// TIA Portal V15.1 export
// export: Created 2024-05-17T05:38:55.5007339Z, ExportSetting WithDefaults, DisplayName Totally Integrated Automation Portal, DisplayVersion V15.1 Update 5, DisplayName TIA Portal Openness, DisplayVersion V15.1 Update 5, DisplayName SINAMICS Startdrive Advanced, DisplayVersion V15.1, DisplayName G130, G150, S120, S150, SINAMICS MV, S210, DisplayVersion V15.1, DisplayName G110M, G120, G120C, G120D, G120P, DisplayVersion V15.1, DisplayName STEP 7 Professional, DisplayVersion V15.1 Update 5, DisplayName STEP 7 Safety, DisplayVersion V15.1, DisplayName WinCC Professional, DisplayVersion V15.1 Update 5, DisplayName SIMATIC Visualization Architect, DisplayVersion V15.1
FUNCTION "209220ZM01Config" : Void   // FC352, FBD
TITLE = 209220ZM01 ModeZone Configuration
{ S7_Optimized_Access := 'FALSE' }
AUTHOR : VCC
VERSION : 0.1
// stored: AutoNumber false, IsIECCheckEnabled false, SetENOAutomatically False, UDAEnableTagReadback false
BEGIN

REGION Network 1: **** 4.2 - Machine Status - Parameters **** Andon
   // Andon Config VCG
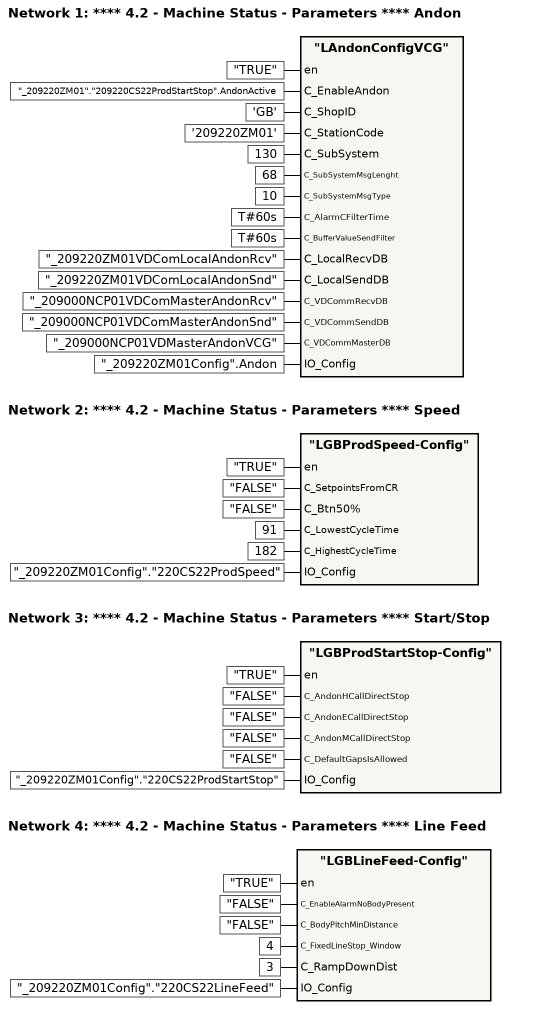
   IF "TRUE" THEN
       "LAndonConfigVCG"(C_EnableAndon := "_209220ZM01"."209220CS22ProdStartStop".AndonActive,
                         C_ShopID := 'GB',
                         C_StationCode := '209220ZM01',
                         C_SubSystem := 130,
                         C_SubSystemMsgLenght := 68,
                         C_SubSystemMsgType := 10,
                         C_AlarmCFilterTime := T#60s,
                         C_BufferValueSendFilter := T#60s,
                         C_LocalRecvDB := "_209220ZM01VDComLocalAndonRcv",
                         C_LocalSendDB := "_209220ZM01VDComLocalAndonSnd",
                         C_VDCommRecvDB := "_209000NCP01VDComMasterAndonRcv",
                         C_VDCommSendDB := "_209000NCP01VDComMasterAndonSnd",
                         C_VDCommMasterDB := "_209000NCP01VDMasterAndonVCG",
                         IO_Config := "_209220ZM01Config".Andon);
   END_IF;
END_REGION

REGION Network 2: **** 4.2 - Machine Status - Parameters **** Speed
   IF "TRUE" THEN
       "LGBProdSpeed-Config"(C_SetpointsFromCR := "FALSE",
                             "C_Btn50%" := "FALSE",
                             C_LowestCycleTime := 91,
                             C_HighestCycleTime := 182,
                             IO_Config := "_209220ZM01Config"."220CS22ProdSpeed");
   END_IF;
END_REGION

REGION Network 3: **** 4.2 - Machine Status - Parameters **** Start/Stop
   IF "TRUE" THEN
       "LGBProdStartStop-Config"(C_AndonHCallDirectStop := "FALSE",
                               C_AndonECallDirectStop := "FALSE",
                               C_AndonMCallDirectStop := "FALSE",
                               C_DefaultGapsIsAllowed := "FALSE",
                               IO_Config := "_209220ZM01Config"."220CS22ProdStartStop");
   END_IF;
END_REGION

REGION Network 4: **** 4.2 - Machine Status - Parameters **** Line Feed
   IF "TRUE" THEN
       "LGBLineFeed-Config"(C_EnableAlarmNoBodyPresent := "FALSE",
                            C_BodyPitchMinDistance := "FALSE",
                            C_FixedLineStop_Window := 4,
                            C_RampDownDist := 3,
                            IO_Config := "_209220ZM01Config"."220CS22LineFeed");
   END_IF;
END_REGION

REGION Network 5: **** 4.2 - Machine Status - Parameters **** Shift Register
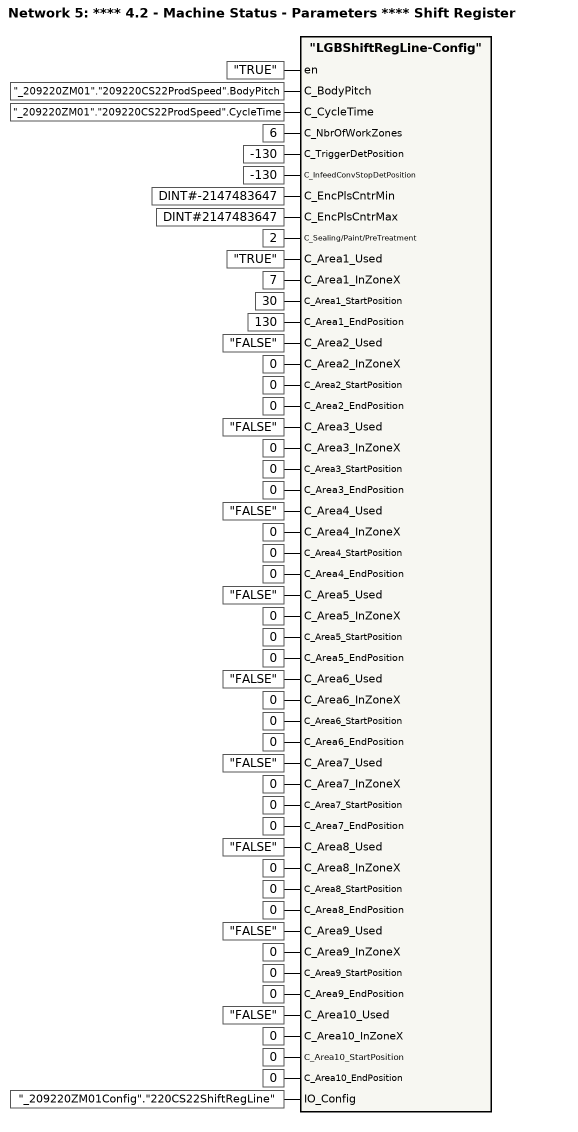
   IF "TRUE" THEN
       "LGBShiftRegLine-Config"(C_BodyPitch := "_209220ZM01"."209220CS22ProdSpeed".BodyPitch,
                               C_CycleTime := "_209220ZM01"."209220CS22ProdSpeed".CycleTime,
                               C_NbrOfWorkZones := 6,
                               C_TriggerDetPosition := -130,
                               C_InfeedConvStopDetPosition := -130,
                               C_EncPlsCntrMin := DINT#-2147483647,
                               C_EncPlsCntrMax := DINT#2147483647,
                               "C_Sealing/Paint/PreTreatment" := 2,
                               C_Area1_Used := "TRUE",
                               C_Area1_InZoneX := 7,
                               C_Area1_StartPosition := 30,
                               C_Area1_EndPosition := 130,
                               C_Area2_Used := "FALSE",
                               C_Area2_InZoneX := 0,
                               C_Area2_StartPosition := 0,
                               C_Area2_EndPosition := 0,
                               C_Area3_Used := "FALSE",
                               C_Area3_InZoneX := 0,
                               C_Area3_StartPosition := 0,
                               C_Area3_EndPosition := 0,
                               C_Area4_Used := "FALSE",
                               C_Area4_InZoneX := 0,
                               C_Area4_StartPosition := 0,
                               C_Area4_EndPosition := 0,
                               C_Area5_Used := "FALSE",
                               C_Area5_InZoneX := 0,
                               C_Area5_StartPosition := 0,
                               C_Area5_EndPosition := 0,
                               C_Area6_Used := "FALSE",
                               C_Area6_InZoneX := 0,
                               C_Area6_StartPosition := 0,
                               C_Area6_EndPosition := 0,
                               C_Area7_Used := "FALSE",
                               C_Area7_InZoneX := 0,
                               C_Area7_StartPosition := 0,
                               C_Area7_EndPosition := 0,
                               C_Area8_Used := "FALSE",
                               C_Area8_InZoneX := 0,
                               C_Area8_StartPosition := 0,
                               C_Area8_EndPosition := 0,
                               C_Area9_Used := "FALSE",
                               C_Area9_InZoneX := 0,
                               C_Area9_StartPosition := 0,
                               C_Area9_EndPosition := 0,
                               C_Area10_Used := "FALSE",
                               C_Area10_InZoneX := 0,
                               C_Area10_StartPosition := 0,
                               C_Area10_EndPosition := 0,
                               IO_Config := "_209220ZM01Config"."220CS22ShiftRegLine");
   END_IF;
END_REGION

REGION Network 6: **** 4.2 - Machine Status - Parameters **** 220CHB21
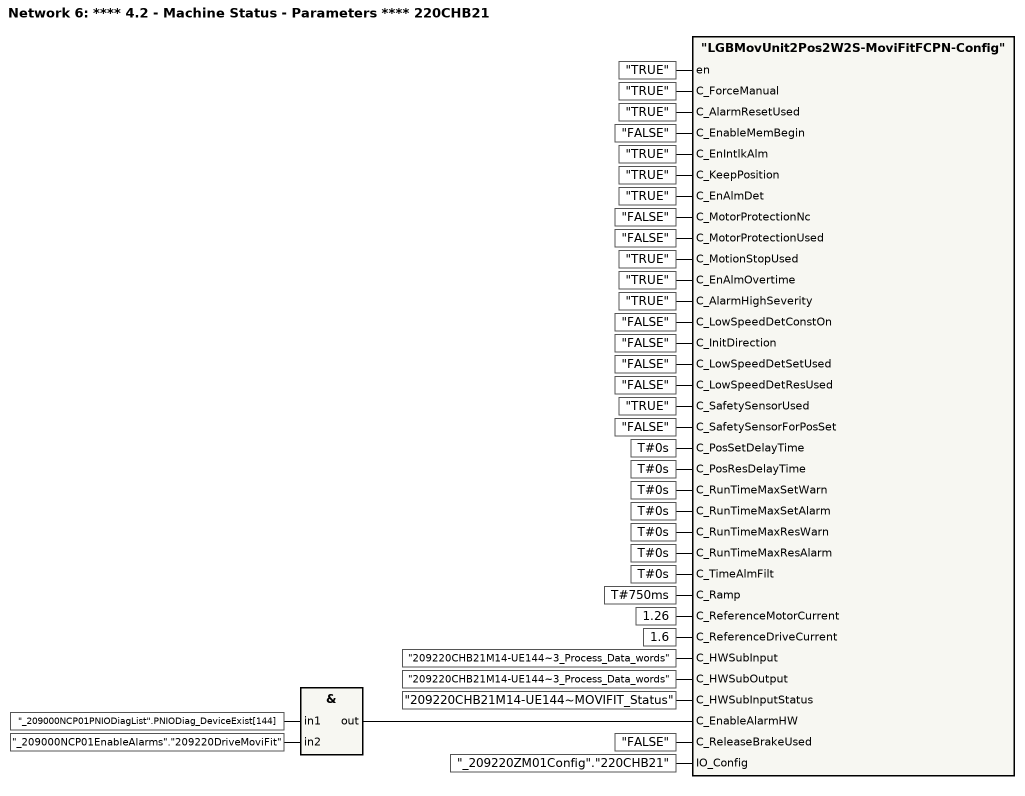
   IF "TRUE" THEN
       "LGBMovUnit2Pos2W2S-MoviFitFCPN-Config"(C_ForceManual := "TRUE",
                               C_AlarmResetUsed := "TRUE",
                               C_EnableMemBegin := "FALSE",
                               C_EnIntlkAlm := "TRUE",
                               C_KeepPosition := "TRUE",
                               C_EnAlmDet := "TRUE",
                               C_MotorProtectionNc := "FALSE",
                               C_MotorProtectionUsed := "FALSE",
                               C_MotionStopUsed := "TRUE",
                               C_EnAlmOvertime := "TRUE",
                               C_AlarmHighSeverity := "TRUE",
                               C_LowSpeedDetConstOn := "FALSE",
                               C_InitDirection := "FALSE",
                               C_LowSpeedDetSetUsed := "FALSE",
                               C_LowSpeedDetResUsed := "FALSE",
                               C_SafetySensorUsed := "TRUE",
                               C_SafetySensorForPosSet := "FALSE",
                               C_PosSetDelayTime := T#0s,
                               C_PosResDelayTime := T#0s,
                               C_RunTimeMaxSetWarn := T#0s,
                               C_RunTimeMaxSetAlarm := T#0s,
                               C_RunTimeMaxResWarn := T#0s,
                               C_RunTimeMaxResAlarm := T#0s,
                               C_TimeAlmFilt := T#0s,
                               C_Ramp := T#750ms,
                               C_ReferenceMotorCurrent := 1.26,
                               C_ReferenceDriveCurrent := 1.6,
                               C_HWSubInput := "209220CHB21M14-UE144~3_Process_Data_words",
                               C_HWSubOutput := "209220CHB21M14-UE144~3_Process_Data_words",
                               C_HWSubInputStatus := "209220CHB21M14-UE144~MOVIFIT_Status",
                               C_EnableAlarmHW := "_209000NCP01PNIODiagList".PNIODiag_DeviceExist[144] AND "_209000NCP01EnableAlarms"."209220DriveMoviFit",
                               C_ReleaseBrakeUsed := "FALSE",
                               IO_Config := "_209220ZM01Config"."220CHB21");
   END_IF;
END_REGION

REGION Network 7: **** 4.2 - Machine Status - Parameters **** 220CR21
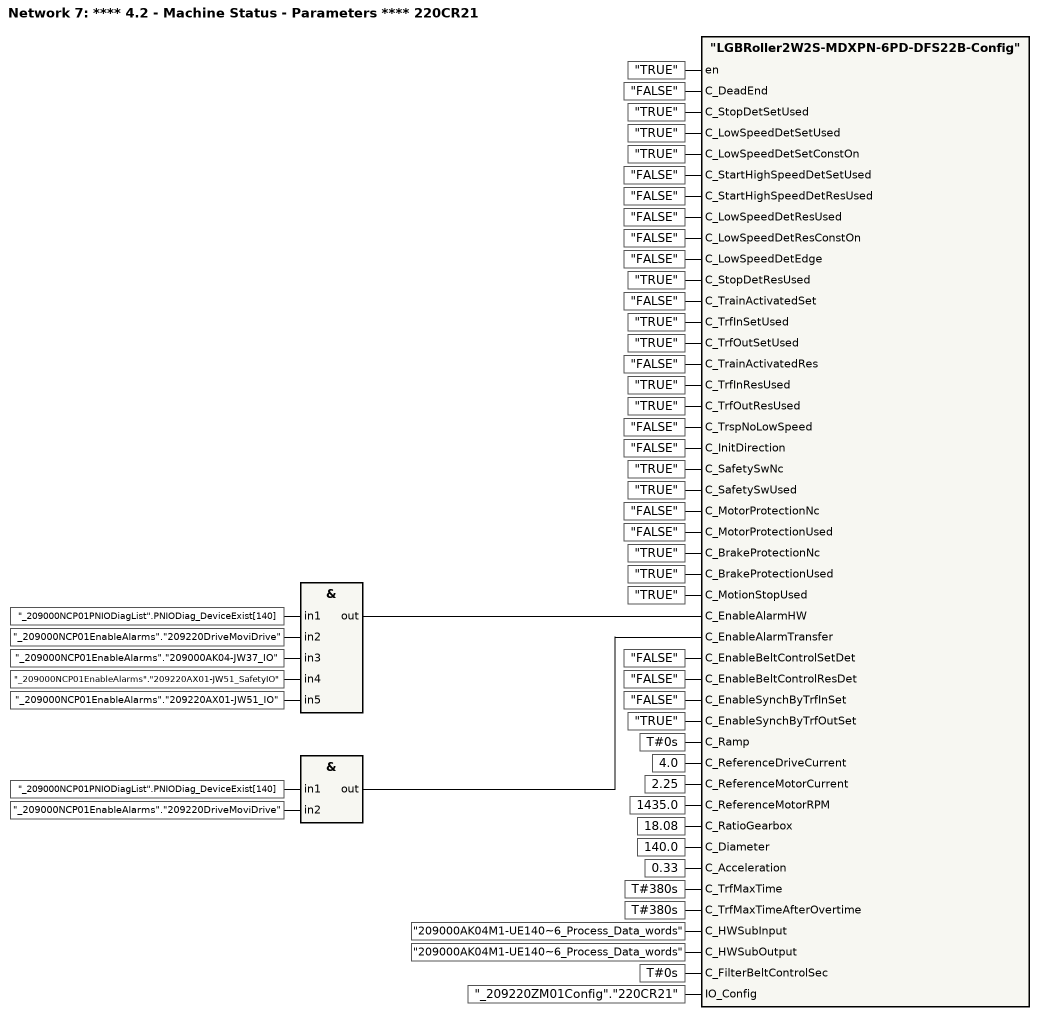
   IF "TRUE" THEN
       "LGBRoller2W2S-MDXPN-6PD-DFS22B-Config"(C_DeadEnd := "FALSE",
                               C_StopDetSetUsed := "TRUE",
                               C_LowSpeedDetSetUsed := "TRUE",
                               C_LowSpeedDetSetConstOn := "TRUE",
                               C_StartHighSpeedDetSetUsed := "FALSE",
                               C_StartHighSpeedDetResUsed := "FALSE",
                               C_LowSpeedDetResUsed := "FALSE",
                               C_LowSpeedDetResConstOn := "FALSE",
                               C_LowSpeedDetEdge := "FALSE",
                               C_StopDetResUsed := "TRUE",
                               C_TrainActivatedSet := "FALSE",
                               C_TrfInSetUsed := "TRUE",
                               C_TrfOutSetUsed := "TRUE",
                               C_TrainActivatedRes := "FALSE",
                               C_TrfInResUsed := "TRUE",
                               C_TrfOutResUsed := "TRUE",
                               C_TrspNoLowSpeed := "FALSE",
                               C_InitDirection := "FALSE",
                               C_SafetySwNc := "TRUE",
                               C_SafetySwUsed := "TRUE",
                               C_MotorProtectionNc := "FALSE",
                               C_MotorProtectionUsed := "FALSE",
                               C_BrakeProtectionNc := "TRUE",
                               C_BrakeProtectionUsed := "TRUE",
                               C_MotionStopUsed := "TRUE",
                               C_EnableAlarmHW := "_209000NCP01PNIODiagList".PNIODiag_DeviceExist[140] AND "_209000NCP01EnableAlarms"."209220DriveMoviDrive" AND "_209000NCP01EnableAlarms"."209000AK04-JW37_IO" AND "_209000NCP01EnableAlarms"."209220AX01-JW51_SafetyIO" AND "_209000NCP01EnableAlarms"."209220AX01-JW51_IO",
                               C_EnableAlarmTransfer := "_209000NCP01PNIODiagList".PNIODiag_DeviceExist[140] AND "_209000NCP01EnableAlarms"."209220DriveMoviDrive",
                               C_EnableBeltControlSetDet := "FALSE",
                               C_EnableBeltControlResDet := "FALSE",
                               C_EnableSynchByTrfInSet := "FALSE",
                               C_EnableSynchByTrfOutSet := "TRUE",
                               C_Ramp := T#0s,
                               C_ReferenceDriveCurrent := 4.0,
                               C_ReferenceMotorCurrent := 2.25,
                               C_ReferenceMotorRPM := 1435.0,
                               C_RatioGearbox := 18.08,
                               C_Diameter := 140.0,
                               C_Acceleration := 0.33,
                               C_TrfMaxTime := T#380s,
                               C_TrfMaxTimeAfterOvertime := T#380s,
                               C_HWSubInput := "209000AK04M1-UE140~6_Process_Data_words",
                               C_HWSubOutput := "209000AK04M1-UE140~6_Process_Data_words",
                               C_FilterBeltControlSec := T#0s,
                               IO_Config := "_209220ZM01Config"."220CR21");
   END_IF;
END_REGION

REGION Network 8: **** 4.2 - Machine Status - Parameters **** 220CS22
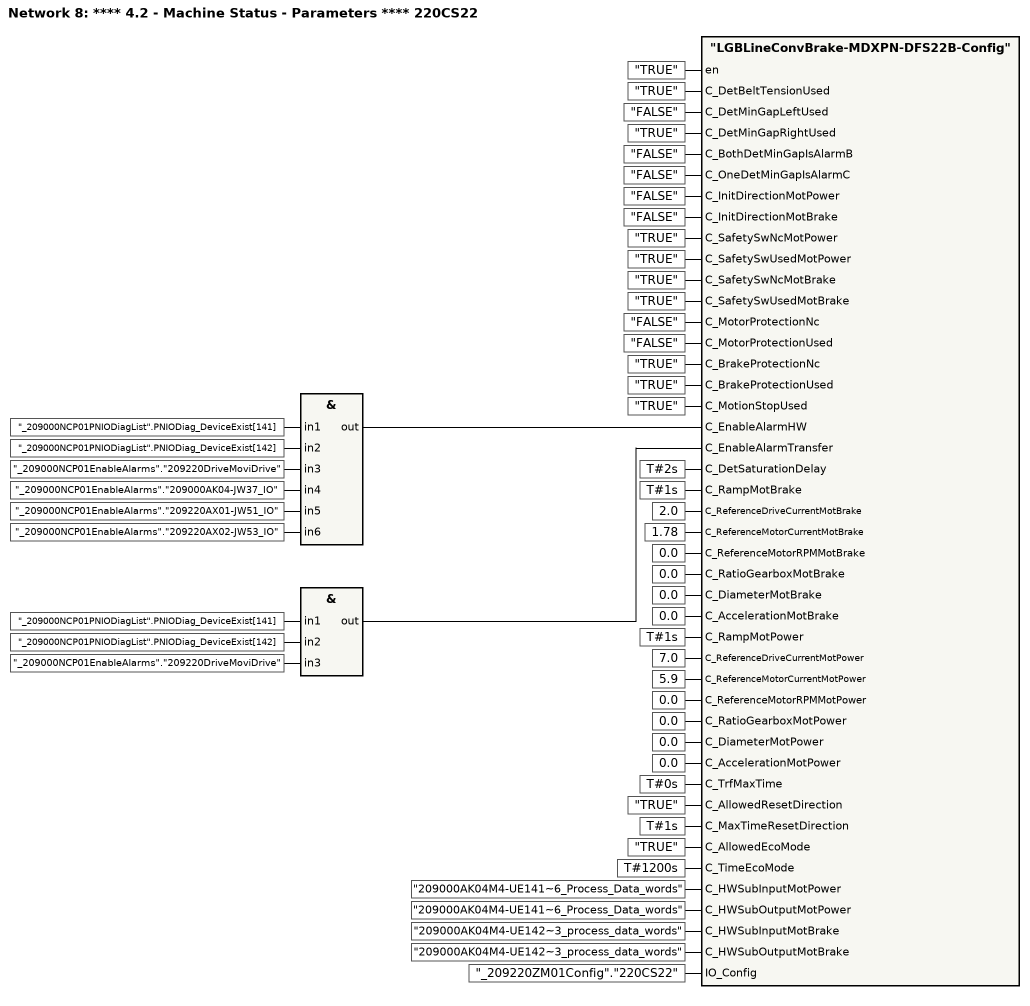
   IF "TRUE" THEN
       "LGBLineConvBrake-MDXPN-DFS22B-Config"(C_DetBeltTensionUsed := "TRUE",
                               C_DetMinGapLeftUsed := "FALSE",
                               C_DetMinGapRightUsed := "TRUE",
                               C_BothDetMinGapIsAlarmB := "FALSE",
                               C_OneDetMinGapIsAlarmC := "FALSE",
                               C_InitDirectionMotPower := "FALSE",
                               C_InitDirectionMotBrake := "FALSE",
                               C_SafetySwNcMotPower := "TRUE",
                               C_SafetySwUsedMotPower := "TRUE",
                               C_SafetySwNcMotBrake := "TRUE",
                               C_SafetySwUsedMotBrake := "TRUE",
                               C_MotorProtectionNc := "FALSE",
                               C_MotorProtectionUsed := "FALSE",
                               C_BrakeProtectionNc := "TRUE",
                               C_BrakeProtectionUsed := "TRUE",
                               C_MotionStopUsed := "TRUE",
                               C_EnableAlarmHW := "_209000NCP01PNIODiagList".PNIODiag_DeviceExist[141] AND "_209000NCP01PNIODiagList".PNIODiag_DeviceExist[142] AND "_209000NCP01EnableAlarms"."209220DriveMoviDrive" AND "_209000NCP01EnableAlarms"."209000AK04-JW37_IO" AND "_209000NCP01EnableAlarms"."209220AX01-JW51_IO" AND "_209000NCP01EnableAlarms"."209220AX02-JW53_IO",
                               C_EnableAlarmTransfer := "_209000NCP01PNIODiagList".PNIODiag_DeviceExist[141] AND "_209000NCP01PNIODiagList".PNIODiag_DeviceExist[142] AND "_209000NCP01EnableAlarms"."209220DriveMoviDrive",
                               C_DetSaturationDelay := T#2s,
                               C_RampMotBrake := T#1s,
                               C_ReferenceDriveCurrentMotBrake := 2.0,
                               C_ReferenceMotorCurrentMotBrake := 1.78,
                               C_ReferenceMotorRPMMotBrake := 0.0,
                               C_RatioGearboxMotBrake := 0.0,
                               C_DiameterMotBrake := 0.0,
                               C_AccelerationMotBrake := 0.0,
                               C_RampMotPower := T#1s,
                               C_ReferenceDriveCurrentMotPower := 7.0,
                               C_ReferenceMotorCurrentMotPower := 5.9,
                               C_ReferenceMotorRPMMotPower := 0.0,
                               C_RatioGearboxMotPower := 0.0,
                               C_DiameterMotPower := 0.0,
                               C_AccelerationMotPower := 0.0,
                               C_TrfMaxTime := T#0s,
                               C_AllowedResetDirection := "TRUE",
                               C_MaxTimeResetDirection := T#1s,
                               C_AllowedEcoMode := "TRUE",
                               C_TimeEcoMode := T#1200s,
                               C_HWSubInputMotPower := "209000AK04M4-UE141~6_Process_Data_words",
                               C_HWSubOutputMotPower := "209000AK04M4-UE141~6_Process_Data_words",
                               C_HWSubInputMotBrake := "209000AK04M4-UE142~3_process_data_words",
                               C_HWSubOutputMotBrake := "209000AK04M4-UE142~3_process_data_words",
                               IO_Config := "_209220ZM01Config"."220CS22");
   END_IF;
END_REGION

REGION Network 9: **** 4.2 - Machine Status - Parameters **** 220CR23
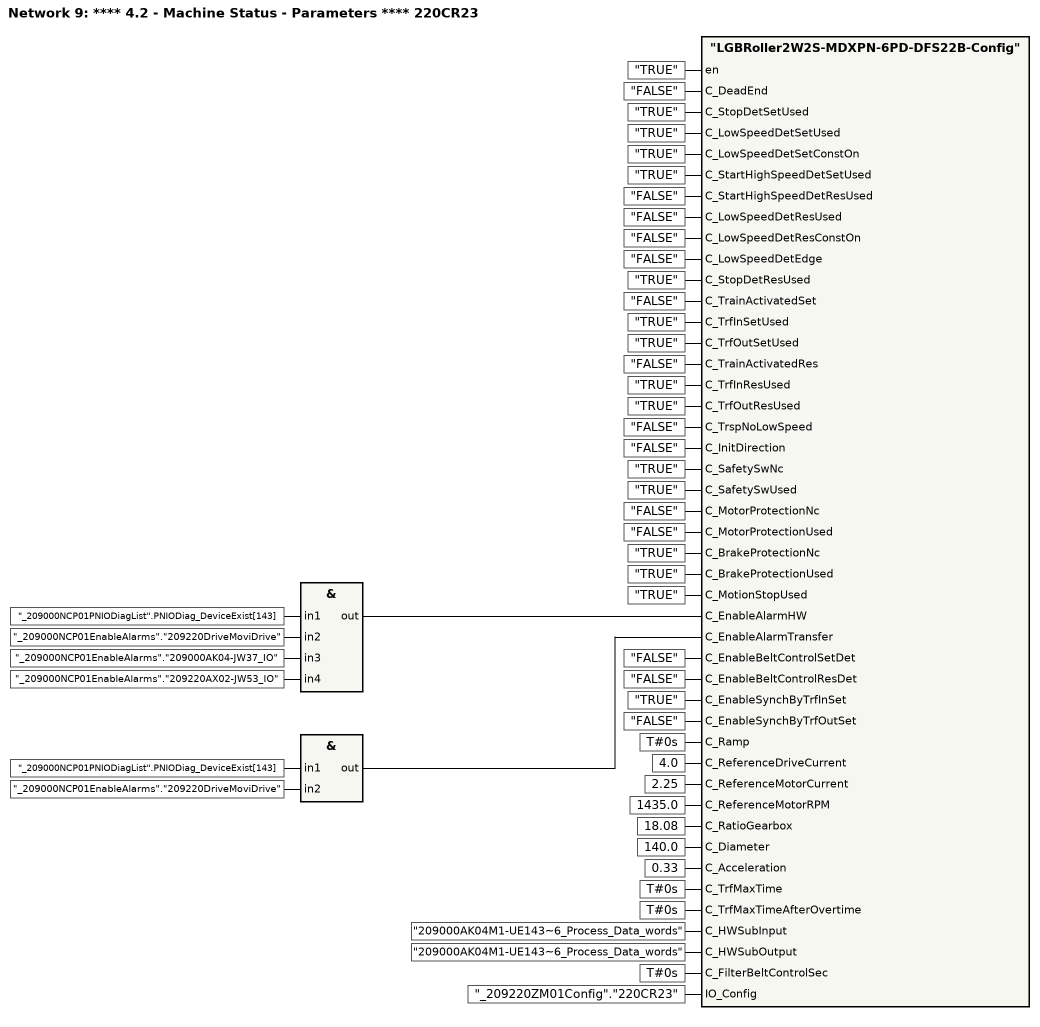
   IF "TRUE" THEN
       "LGBRoller2W2S-MDXPN-6PD-DFS22B-Config"(C_DeadEnd := "FALSE",
                               C_StopDetSetUsed := "TRUE",
                               C_LowSpeedDetSetUsed := "TRUE",
                               C_LowSpeedDetSetConstOn := "TRUE",
                               C_StartHighSpeedDetSetUsed := "TRUE",
                               C_StartHighSpeedDetResUsed := "FALSE",
                               C_LowSpeedDetResUsed := "FALSE",
                               C_LowSpeedDetResConstOn := "FALSE",
                               C_LowSpeedDetEdge := "FALSE",
                               C_StopDetResUsed := "TRUE",
                               C_TrainActivatedSet := "FALSE",
                               C_TrfInSetUsed := "TRUE",
                               C_TrfOutSetUsed := "TRUE",
                               C_TrainActivatedRes := "FALSE",
                               C_TrfInResUsed := "TRUE",
                               C_TrfOutResUsed := "TRUE",
                               C_TrspNoLowSpeed := "FALSE",
                               C_InitDirection := "FALSE",
                               C_SafetySwNc := "TRUE",
                               C_SafetySwUsed := "TRUE",
                               C_MotorProtectionNc := "FALSE",
                               C_MotorProtectionUsed := "FALSE",
                               C_BrakeProtectionNc := "TRUE",
                               C_BrakeProtectionUsed := "TRUE",
                               C_MotionStopUsed := "TRUE",
                               C_EnableAlarmHW := "_209000NCP01PNIODiagList".PNIODiag_DeviceExist[143] AND "_209000NCP01EnableAlarms"."209220DriveMoviDrive" AND "_209000NCP01EnableAlarms"."209000AK04-JW37_IO" AND "_209000NCP01EnableAlarms"."209220AX02-JW53_IO",
                               C_EnableAlarmTransfer := "_209000NCP01PNIODiagList".PNIODiag_DeviceExist[143] AND "_209000NCP01EnableAlarms"."209220DriveMoviDrive",
                               C_EnableBeltControlSetDet := "FALSE",
                               C_EnableBeltControlResDet := "FALSE",
                               C_EnableSynchByTrfInSet := "TRUE",
                               C_EnableSynchByTrfOutSet := "FALSE",
                               C_Ramp := T#0s,
                               C_ReferenceDriveCurrent := 4.0,
                               C_ReferenceMotorCurrent := 2.25,
                               C_ReferenceMotorRPM := 1435.0,
                               C_RatioGearbox := 18.08,
                               C_Diameter := 140.0,
                               C_Acceleration := 0.33,
                               C_TrfMaxTime := T#0s,
                               C_TrfMaxTimeAfterOvertime := T#0s,
                               C_HWSubInput := "209000AK04M1-UE143~6_Process_Data_words",
                               C_HWSubOutput := "209000AK04M1-UE143~6_Process_Data_words",
                               C_FilterBeltControlSec := T#0s,
                               IO_Config := "_209220ZM01Config"."220CR23");
   END_IF;
END_REGION

REGION Network 10: **** 4.2 - Machine Status - Parameters **** 220ASH01
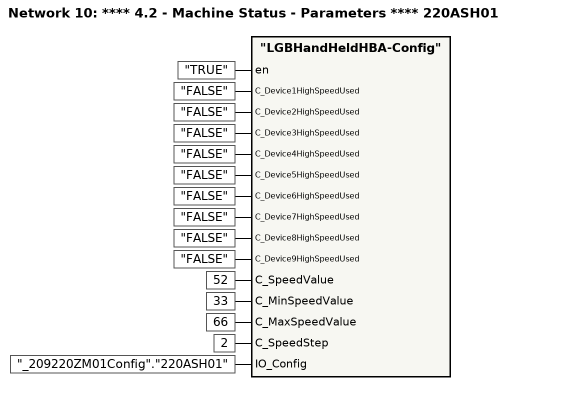
   IF "TRUE" THEN
       "LGBHandHeldHBA-Config"(C_Device1HighSpeedUsed := "FALSE",
                               C_Device2HighSpeedUsed := "FALSE",
                               C_Device3HighSpeedUsed := "FALSE",
                               C_Device4HighSpeedUsed := "FALSE",
                               C_Device5HighSpeedUsed := "FALSE",
                               C_Device6HighSpeedUsed := "FALSE",
                               C_Device7HighSpeedUsed := "FALSE",
                               C_Device8HighSpeedUsed := "FALSE",
                               C_Device9HighSpeedUsed := "FALSE",
                               C_SpeedValue := 52,
                               C_MinSpeedValue := 33,
                               C_MaxSpeedValue := 66,
                               C_SpeedStep := 2,
                               IO_Config := "_209220ZM01Config"."220ASH01");
   END_IF;
END_REGION
END_FUNCTION
